// TIA Portal V19 export
DATA_BLOCK "CallEquipment_DB"   // DB16
AUTHOR : Siemens_FA_SUP
// stored: InstanceOfName Unit2.EM3.CallEquipment, InstanceOfType FB, Namespace Unit2.EM3
"Unit2.EM3.CallEquipment"
   // VAR_IN_OUT
   //    unitStatus : "LAF_typeUnitStatus";
   //    unitAlarmDB : "LAF_typeAlarms";
   //    emFeedback : "LUC_typeEmFeedback";
   // END_VAR
   // VAR
   //    statUnitStatus { ExternalWritable := 'False'} : "LAF_typeUnitStatus";
   //    instJobExecute { ExternalWritable := 'False'} : "LAF_SelectJob";
   //    instJobStopping { ExternalWritable := 'False'; S7_SetPoint := 'True'} : "LAF_SelectJob";
   //    instJobStarting { ExternalWritable := 'False'; S7_SetPoint := 'True'} : "LAF_SelectJob";
   //    instJobHolding { ExternalWritable := 'False'; S7_SetPoint := 'True'} : "LAF_SelectJob";
   //    instJobUnHolding { ExternalWritable := 'False'; S7_SetPoint := 'True'} : "LAF_SelectJob";
   //    instJobReseting { ExternalWritable := 'False'; S7_SetPoint := 'True'} : "LAF_SelectJob";
   //    instSequence { ExternalWritable := 'False'} : "Unit2.EM3.Sequence";
   //    instManageBitAlarms { ExternalWritable := 'False'} : "LAF_ManageBitAlarms";
   //    instCmReset { ExternalWritable := 'False'} : "Unit2.EM3.EXCHANGETRAY_CmResetOperator";
   //    instCm1SV112_Constraint1_Axis { ExternalWritable := 'False'} : "LBC_AxisSimpleControl";
   //    instCm2SV113_Constraint2_Axis { ExternalWritable := 'False'; S7_SetPoint := 'True'} : "LBC_AxisSimpleControl";
   //    instCm3SV115_Screw1_Axis { ExternalWritable := 'False'} : "LEXCHANGETRAY_SimpleAxis";
   //    instCm4SV116_Screw2_Axis { ExternalWritable := 'False'; S7_SetPoint := 'True'} : "LEXCHANGETRAY_SimpleAxis";
   //    instcm10SignalTM { ExternalWritable := 'False'; S7_SetPoint := 'True'} : "LEXCHANGETRAY_U2Em3SingleTM";
   //    instCm6SlideCylinder1 { ExternalWritable := 'False'; S7_SetPoint := 'True'} : "LEXCHANGETRAY_Cylinder";
   //    instCm7hookClawCylinder1 { ExternalWritable := 'False'; S7_SetPoint := 'True'} : "LEXCHANGETRAY_Cylinder";
   //    instCm8SlideCylinder2 { ExternalWritable := 'False'; S7_SetPoint := 'True'} : "LEXCHANGETRAY_Cylinder";
   //    instCm9hookClawCylinder2 { ExternalWritable := 'False'; S7_SetPoint := 'True'} : "LEXCHANGETRAY_Cylinder";
   //    instCm11PressureGuarge { ExternalWritable := 'False'} : "LEXCHANGETRAY_PressureGaugeRs485";
   //    statLstUnitMode { ExternalWritable := 'False'; S7_SetPoint := 'True'} : DInt;
   //    getValue_sp3_1 { ExternalWritable := 'False'} : Array[0..2] of DInt;
   //    getValue_sp3_2 { ExternalWritable := 'False'} : Array[0..2] of DInt;
   //    step_rs485 { ExternalWritable := 'False'} : Int;
   //    statWriteMode { ExternalWritable := 'False'} : Bool;
   // END_VAR
BEGIN
END_DATA_BLOCK
